(* IEC 61131-3 sources: programs/VI-54/VI-54_20171205/VI-54_20171205/Stations/Screen/LseClass170718/Class/GetOSVer, 1 file *)

(* ---- GetOSVer.st ---- *)
(*!
<Class
	Name               = "GetOSVer"
	Revision           = "0.0"
	RealtimeTask       = "false"
	CyclicTask         = "false"
	BackgroundTask     = "false"
	Sigmatek           = "false"
	OSInterface        = "false"
	HighPriority       = "false"
	Automatic          = "false"
	UpdateMode         = "Prescan"
	SharedCommandTable = "true"
	Objectsize         = "(630,240)">
	<Channels>
		<Server Name="ClassSvr" Visualized="false" Initialize="false" WriteProtected="true" Retentive="false"/>
		<Client Name="toGraphic" Required="false" Internal="false"/>
		<Client Name="toOSString" Required="true" Internal="false"/>
		<Client Name="toResString" Required="true" Internal="false"/>
	</Channels>
</Class>
*)
GetOSVer : CLASS
  //Servers:
	ClassSvr 	: SvrChCmd_DINT;
  //Clients:
	toOSString 	: CltChCmd_String;
	toGraphic 	: CltChCmd_Graphic;
	toResString 	: CltChCmd_String;
  //Variables:
  //Functions:

	FUNCTION VIRTUAL GLOBAL Init;
  //Tables:
	FUNCTION @STD
		VAR_OUTPUT
			ret_code	: CONFSTATES;
		END_VAR;
	FUNCTION GLOBAL TAB @CT_;
END_CLASS;

#pragma usingLtd Graphic
#pragma usingLtd String

FUNCTION VIRTUAL GLOBAL GetOSVer::Init
  VAR
    OSVersion : ARRAY[0..11] of CHAR;
    OS1       : UDINT;
    OS2       : UDINT;
    OS3       : UDINT;
    Screen    : _ROOM;
    ScreenStr : ARRAY[0..11] of CHAR;
    Length    : UDINT;
  END_VAR

  if _firstscan = 1 then

    toGraphic.GetScreenSize(#Screen);
    DtoA(#ScreenStr[0],Screen.xy2.x + 1,16#0800,sizeof(_ASCII));
    StrCat(#ScreenStr[0],sizeof(_ASCII)," x ",sizeof(_ASCII));
    Length := StrLen(#ScreenStr[0],sizeof(_ASCII));
    DtoA(#ScreenStr[Length],Screen.xy2.y + 1,16#0800,sizeof(_ASCII));
    toResString.WriteDataOff(udLen := 12, udOff := 0, #ScreenStr[0]);

    OS1 := _RtosVersion shr 12 and 16#0000000F;
		OS2 := _RtosVersion shr 8  and 16#0000000F;
		OS3 := _RtosVersion        and 16#000000FF;

    DtoA(#OSVersion[0],to_DINT(OS1),0x0102,sizeof(_ASCII));
    OSVersion[2] := '.';
    DtoA(#OSVersion[3],to_DINT(OS2),0x0102,sizeof(_ASCII));
    OSVersion[5] := '.';
    DtoA(#OSVersion[6],to_DINT(OS3),0x0103,sizeof(_ASCII));

		toOSString.WriteDataOff(udLen := 12, udOff := 0, #OSVersion[0]);
	end_if;
END_FUNCTION
